Omron CX-Programmer project NewProject (CX-Programmer 8.01)

# PLC NewPLC1: CP1L M

## Program Sewage_Treatment (cyclic task 0)
Local symbols
HLS_1 0.02 BOOL  ; High Level Switch 1
HLS_2 0.04 BOOL  ; High Level Switch 2
HLS_3 0.06 BOOL  ; High Level Switch 3
HLS_4 0.08 BOOL  ; High Level Switch 4
LLS_1 0.03 BOOL  ; Low Level Switch 1
LLS_2 0.05 BOOL  ; Low Level Switch 2
LLS_3 0.07 BOOL  ; Low Level Switch 3
LLS_4 0.09 BOOL  ; Low Level Switch 4
Motor_A 100.04 BOOL  ; Pump 1
Motor_B 100.05 BOOL  ; Pump 2
Motor_C 100.06 BOOL  ; Pump 3
Motor_D 100.07 BOOL  ; Fan 1
Motor_E 101.00 BOOL  ; Fan 2
Preliminary_State W0.01 BOOL  ; Preliminary Screening
Primary_State W0.02 BOOL  ; Primary Treatment
Secondary_State_1 W0.03 BOOL  ; Secondary Treatment 1
Secondary_State_2 W0.04 BOOL  ; Secondary Treatment 2
Solenoid_A 100.00 BOOL  ; Valve 1
Solenoid_B 100.01 BOOL  ; Valve 2
Solenoid_C 100.02 BOOL  ; Valve 3
Solenoid_D 100.03 BOOL  ; Valve 4
Start_PB 0.00 BOOL  ; Start
Stop_PB 0.01 BOOL  ; Emergency Stop
Stopped_State W0.00 BOOL  ; Stopped
Tertiary_State W0.05 BOOL  ; Tertiary Treatment

### Section Initialization

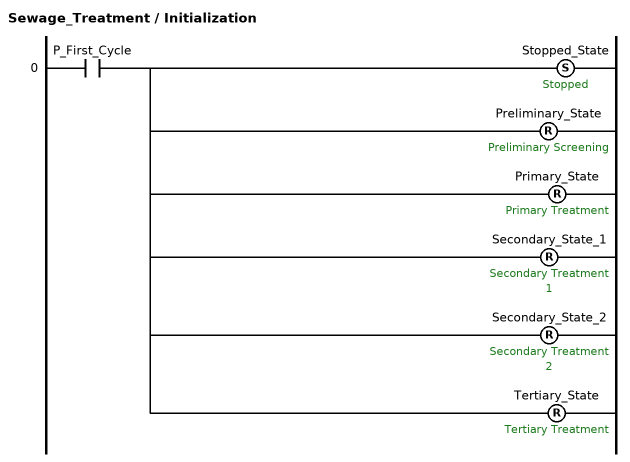
; rung 0
LD P_First_Cycle
SET Stopped_State  ; Stopped
RSET Preliminary_State  ; Preliminary Screening
RSET Primary_State  ; Primary Treatment
RSET Secondary_State_1  ; Secondary Treatment 1
RSET Secondary_State_2  ; Secondary Treatment 2
RSET Tertiary_State  ; Tertiary Treatment

### Section Stopped

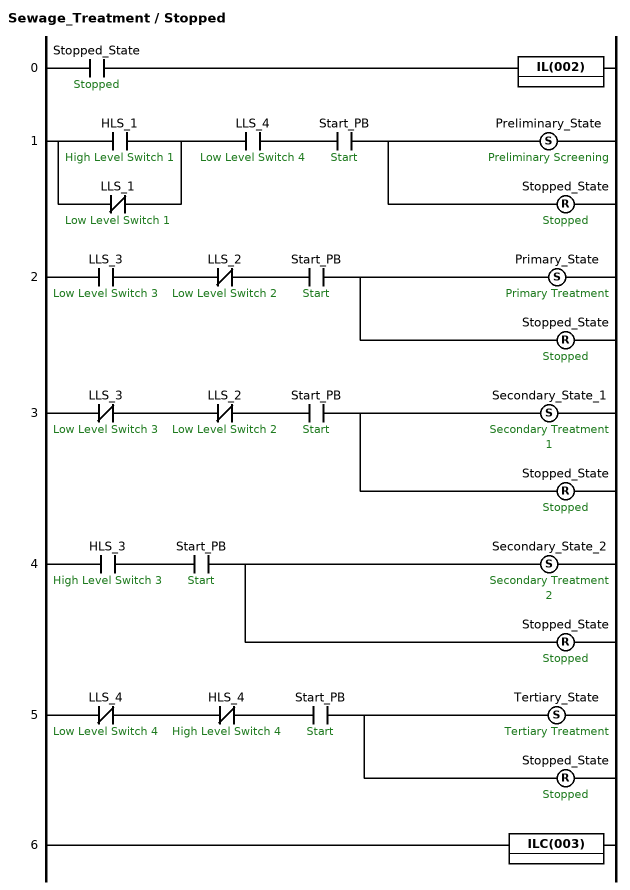
; rung 0
LD Stopped_State  ; Stopped
IL(002)
; rung 1
LD HLS_1  ; High Level Switch 1
ORNOT LLS_1  ; Low Level Switch 1
AND LLS_4  ; Low Level Switch 4
AND Start_PB  ; Start
SET Preliminary_State  ; Preliminary Screening
RSET Stopped_State  ; Stopped
; rung 2
LD LLS_3  ; Low Level Switch 3
ANDNOT LLS_2  ; Low Level Switch 2
AND Start_PB  ; Start
SET Primary_State  ; Primary Treatment
RSET Stopped_State  ; Stopped
; rung 3
LDNOT LLS_3  ; Low Level Switch 3
ANDNOT LLS_2  ; Low Level Switch 2
AND Start_PB  ; Start
SET Secondary_State_1  ; Secondary Treatment 1
RSET Stopped_State  ; Stopped
; rung 4
LD HLS_3  ; High Level Switch 3
AND Start_PB  ; Start
SET Secondary_State_2  ; Secondary Treatment 2
RSET Stopped_State  ; Stopped
; rung 5
LDNOT LLS_4  ; Low Level Switch 4
ANDNOT HLS_4  ; High Level Switch 4
AND Start_PB  ; Start
SET Tertiary_State  ; Tertiary Treatment
RSET Stopped_State  ; Stopped
; rung 6
ILC(003)

### Section Preliminary

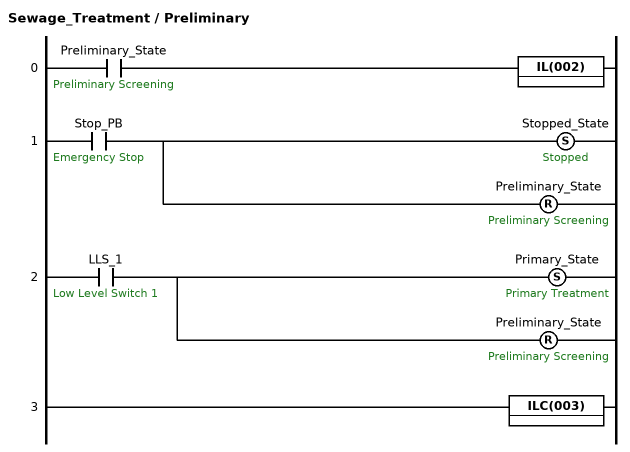
; rung 0
LD Preliminary_State  ; Preliminary Screening
IL(002)
; rung 1
LD Stop_PB  ; Emergency Stop
SET Stopped_State  ; Stopped
RSET Preliminary_State  ; Preliminary Screening
; rung 2
LD LLS_1  ; Low Level Switch 1
SET Primary_State  ; Primary Treatment
RSET Preliminary_State  ; Preliminary Screening
; rung 3
ILC(003)

### Section Primary

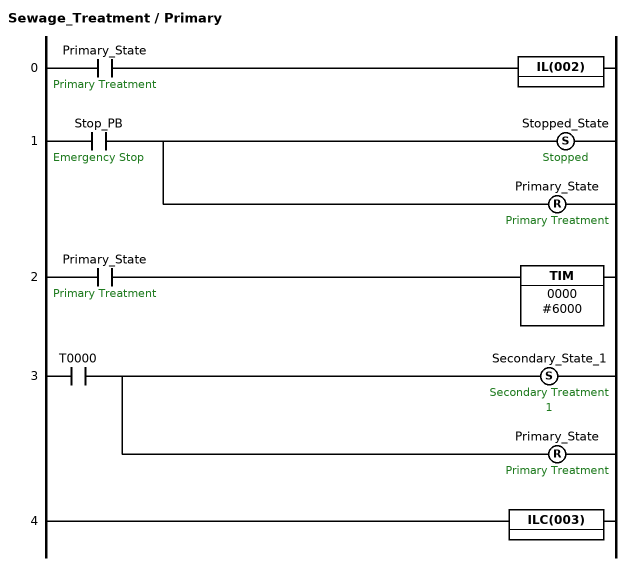
; rung 0
LD Primary_State  ; Primary Treatment
IL(002)
; rung 1
LD Stop_PB  ; Emergency Stop
SET Stopped_State  ; Stopped
RSET Primary_State  ; Primary Treatment
; rung 2
LD Primary_State  ; Primary Treatment
TIM 0000 #6000
; rung 3
LD T0000
SET Secondary_State_1  ; Secondary Treatment 1
RSET Primary_State  ; Primary Treatment
; rung 4
ILC(003)

### Section Secondary_I

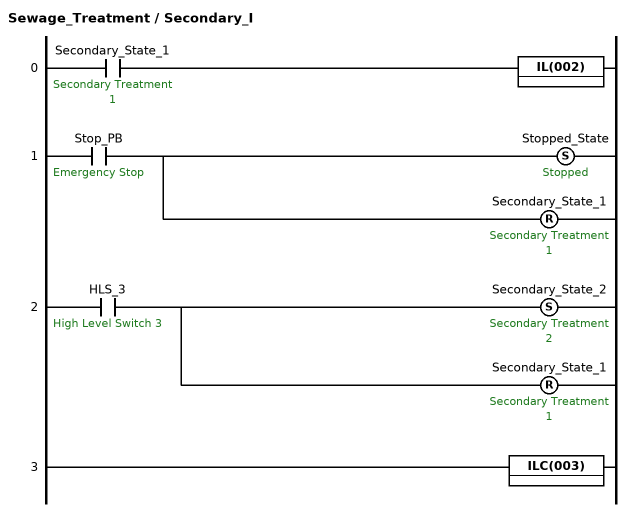
; rung 0
LD Secondary_State_1  ; Secondary Treatment 1
IL(002)
; rung 1
LD Stop_PB  ; Emergency Stop
SET Stopped_State  ; Stopped
RSET Secondary_State_1  ; Secondary Treatment 1
; rung 2
LD HLS_3  ; High Level Switch 3
SET Secondary_State_2  ; Secondary Treatment 2
RSET Secondary_State_1  ; Secondary Treatment 1
; rung 3
ILC(003)

### Section Secondary_II

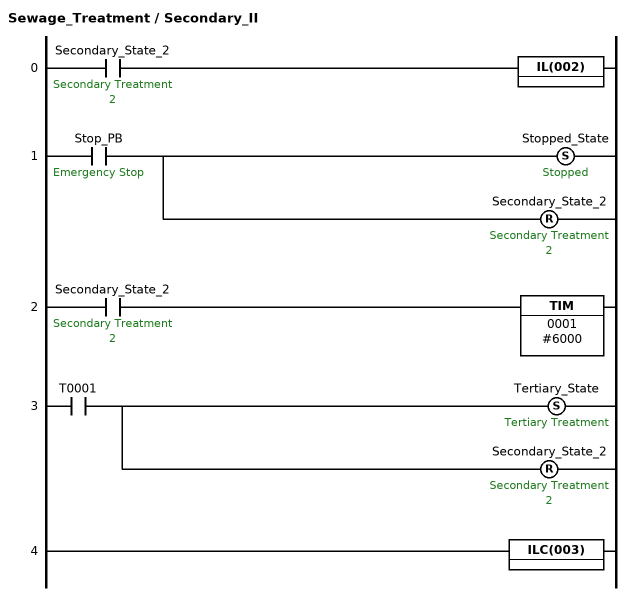
; rung 0
LD Secondary_State_2  ; Secondary Treatment 2
IL(002)
; rung 1
LD Stop_PB  ; Emergency Stop
SET Stopped_State  ; Stopped
RSET Secondary_State_2  ; Secondary Treatment 2
; rung 2
LD Secondary_State_2  ; Secondary Treatment 2
TIM 0001 #6000
; rung 3
LD T0001
SET Tertiary_State  ; Tertiary Treatment
RSET Secondary_State_2  ; Secondary Treatment 2
; rung 4
ILC(003)

### Section Tertiary

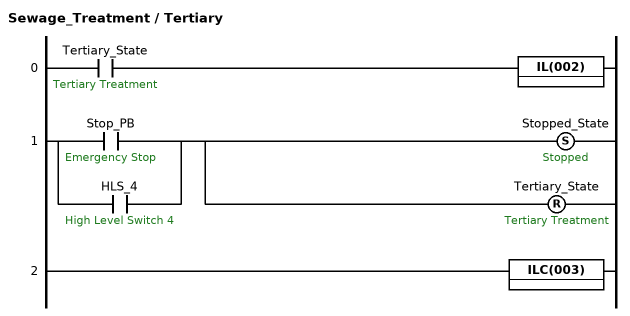
; rung 0
LD Tertiary_State  ; Tertiary Treatment
IL(002)
; rung 1
LD Stop_PB  ; Emergency Stop
OR HLS_4  ; High Level Switch 4
SET Stopped_State  ; Stopped
RSET Tertiary_State  ; Tertiary Treatment
; rung 2
ILC(003)

### Section Outputs

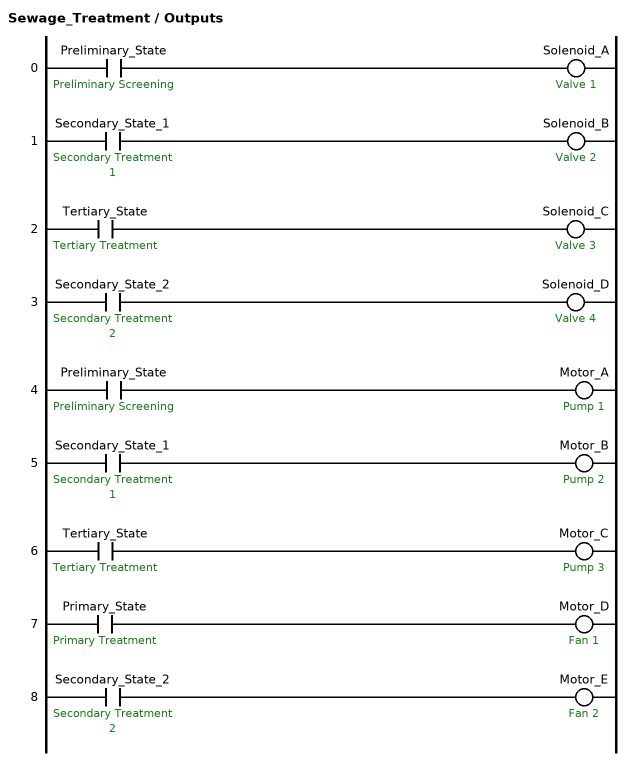
; rung 0
LD Preliminary_State  ; Preliminary Screening
OUT Solenoid_A  ; Valve 1
; rung 1
LD Secondary_State_1  ; Secondary Treatment 1
OUT Solenoid_B  ; Valve 2
; rung 2
LD Tertiary_State  ; Tertiary Treatment
OUT Solenoid_C  ; Valve 3
; rung 3
LD Secondary_State_2  ; Secondary Treatment 2
OUT Solenoid_D  ; Valve 4
; rung 4
LD Preliminary_State  ; Preliminary Screening
OUT Motor_A  ; Pump 1
; rung 5
LD Secondary_State_1  ; Secondary Treatment 1
OUT Motor_B  ; Pump 2
; rung 6
LD Tertiary_State  ; Tertiary Treatment
OUT Motor_C  ; Pump 3
; rung 7
LD Primary_State  ; Primary Treatment
OUT Motor_D  ; Fan 1
; rung 8
LD Secondary_State_2  ; Secondary Treatment 2
OUT Motor_E  ; Fan 2

### Section END
; rung 0
END(001)